FUNCTION_BLOCK  FB_SysLogMsgListener  EXTENDS FB_ListenerBase2
VAR
    Json          : FB_JsonDomParser; 		//Parse JSON attribute of messages
     JsonAttribute : STRING(10000);    		//Holds JSON attribute
     hr            : HRESULT;         		//Signals JSON attribute was successfully read
    ipListener    : I_SysLogListener; 	//Receives callback once message is processed
	
	fbRequestEventText : FB_RequestEventText;
	{attribute 'TcEncoding':='UTF-8'}
	sLastMessageText : STRING;
	
END_VAR

PROPERTY Listener : I_SysLogListener
SET
ipListener := Listener;
END_SET
END_PROPERTY

METHOD OnMessageSent : Tc3_EventLogger.HRESULT
VAR_INPUT
    fbEvent 			: REFERENCE TO FB_TcEvent;
END_VAR

VAR
    message      		: ST_SysLogMessages;
    jsonDocument 		: SJsonValue;
    jsonProperty 		: SJsonValue;
	
	hasMember 			: BOOL;
END_VAR
hr := fbEvent.GetJsonAttribute(JsonAttribute, SIZEOF(JsonAttribute));

IF ( SUCCEEDED(hr) ) THEN
    jsonDocument := json.ParseDocument(JsonAttribute);

    IF ( json.HasMember(jsonDocument, 'Timestamp') ) THEN
        jsonProperty      := json.FindMember(JsonDocument, 'Timestamp');
        message.timestamp := json.GetString(JsonProperty);
    END_IF

    IF ( json.HasMember(jsonDocument, 'Message') ) THEN
        jsonProperty    := json.FindMember(jsonDocument, 'Message');
        message.message := json.GetString(jsonProperty);
    END_IF
	
	IF ( json.HasMember(jsonDocument, 'LogLevel') ) THEN
        jsonProperty      := json.FindMember(jsonDocument, 'LogLevel');
        message.logLevel := json.GetUint(jsonProperty);
    END_IF
	
    IF ( json.HasMember(jsonDocument, 'Source') ) THEN
        jsonProperty   := json.FindMember(jsonDocument, 'Source');
        message.Source := json.GetString(jsonProperty);
    END_IF

    IF ( json.HasMember(jsonDocument, 'Context') ) THEN
        jsonProperty    := json.FindMember(jsonDocument, 'Context');
        message.Context := json.GetString(jsonProperty);
    END_IF

    IF ( json.HasMember(jsonDocument, 'ScanCount') ) THEN
        jsonProperty      := json.FindMember(jsonDocument, 'ScanCount');
        message.ScanCount := json.GetUint(jsonProperty);
    END_IF

    IF ( json.HasMember(jsonDocument, 'Flags') ) THEN
        jsonProperty  := json.FindMember(jsonDocument, 'Flags');
        message.Flags := json.GetUint(jsonProperty);
    END_IF
	
    IF ( json.HasMember(jsonDocument, 'ExtendedInfo') ) THEN
        jsonProperty := json.FindMember(jsonDocument, 'ExtendedInfo');
        message.Json := json.GetString(jsonProperty);
    END_IF


    IF ( ipListener <> 0 ) THEN
        //Notify listener of message data
        ipListener.OnTraceReceived(Message);
    END_IF
END_IF

OnMessageSent := S_OK; // in order to receive more callbacks (Set <> S_OK in order to cancel the callbacks for this program cycle.)
END_METHOD

END_FUNCTION_BLOCK

(* stored: Version 1.1.0.1
   POU FB_SysLogMsgListener: Id {0360203c-1ba6-41bf-8e19-b9bc785da99e}, SpecialFunc None
   Property Listener: Id {e04ea468-0d95-4888-ba76-4a9c305f0ea9}
   Set Set: Id {950bc0e2-707f-40c3-b5ae-1275deac7127}
   Method OnMessageSent: Id {46fa173d-841d-44a4-9b56-28528074126a} *)
